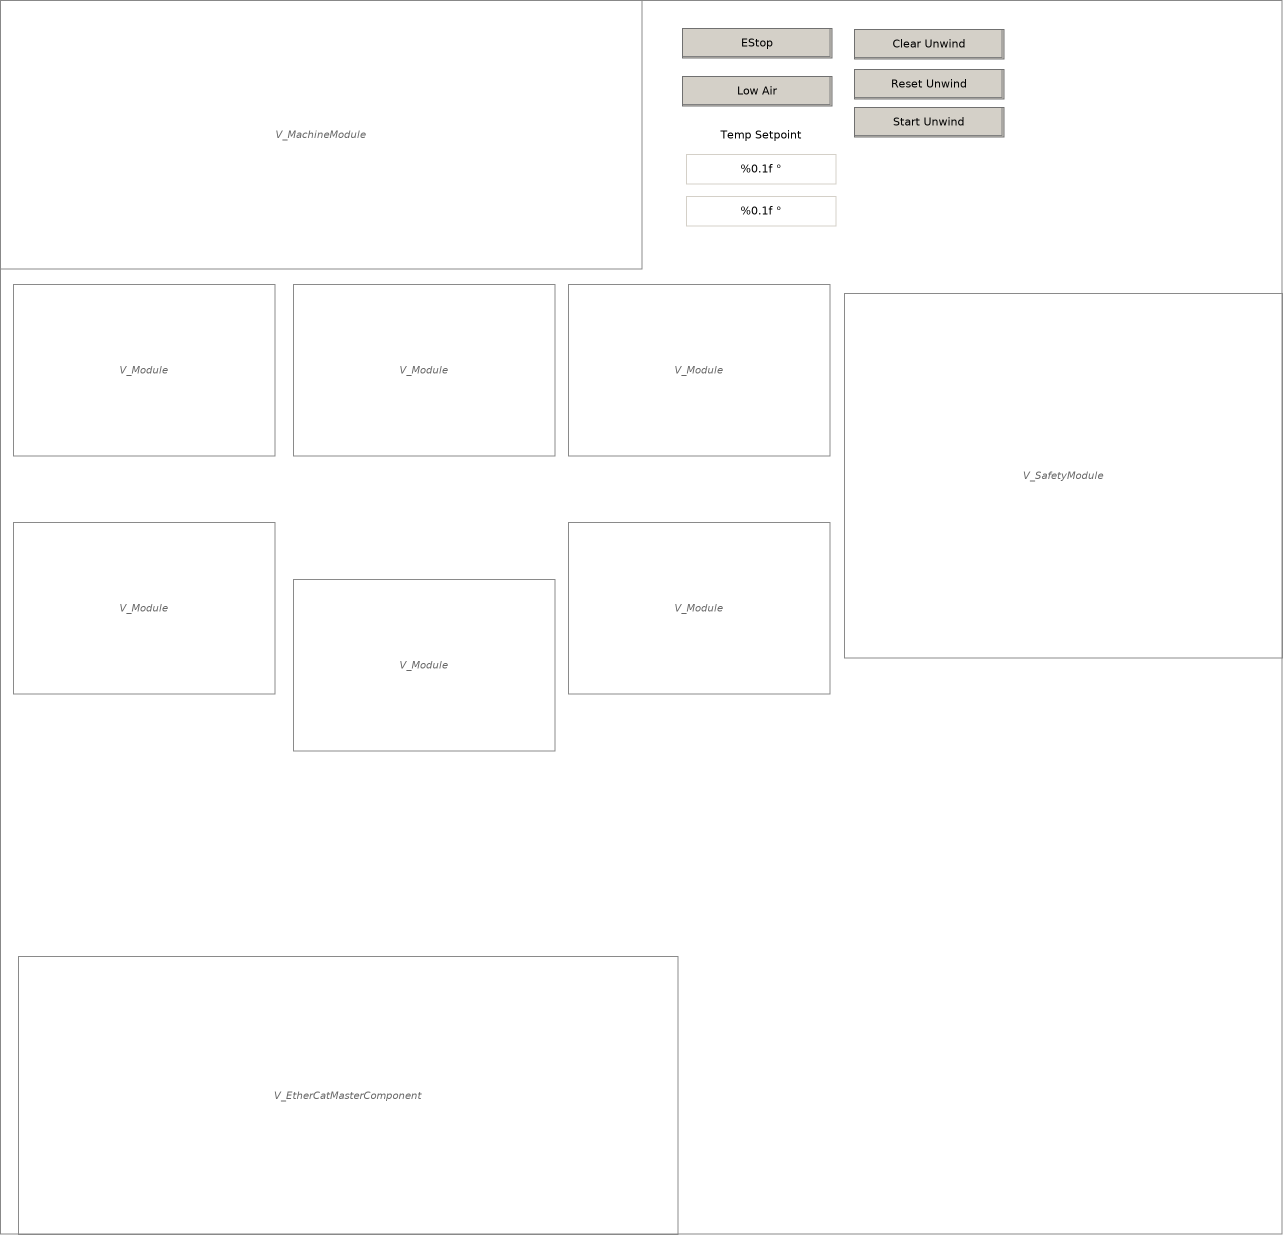
VISUALIZATION V_Main  // 1283x1235
    Frame (0,0 642x269)
        shows V_MachineModule(HMI := MAIN.Machine.PackMLBaseModule_HMI)
    Frame (568,284 262x172)
        shows V_Module(HMI := MAIN.Machine.Station_4.PackMLBaseModule_HMI)
    Frame (568,522 262x172)
        shows V_Module(HMI := MAIN.Machine.Station_5.PackMLBaseModule_HMI)
    Button (682,28 150x30), "EStop"
        toggle MAIN.Machine.EstopInput
    Button (682,76 150x30), "Low Air"
        toggle MAIN.Machine.LowAirInput
    Textfield (686,154 150x30), "%0.1f °", text variable: MAIN.Machine.Sealer.SealBar._SetTemperature
        OnMouseDown: write the text variable via VisuDialogs.Numpad, min 20, max 400, title 'Sealer Bar Temp Setpoint', format %0.1f
    Label (686,120 150x30), "Temp Setpoint"
    Textfield (686,196 150x30), "%0.1f °", text variable: MAIN.Machine.Sealer.SealBar._ActualTemperature
    Button (854,29 150x30), "Clear Unwind"
        OnMouseClick: execute { MAIN.Machine.unwind.PackMLBaseModule_HMI.Command.State := E_PMLCommand.ePMLCommand_Clear; }
    Button (854,69 150x30), "Reset Unwind"
        OnMouseClick: execute { MAIN.Machine.unwind.PackMLBaseModule_HMI.Command.State := E_PMLCommand.ePMLCommand_Reset; }
    Button (854,107 150x30), "Start Unwind"
        OnMouseClick: execute { MAIN.Machine.unwind.PackMLBaseModule_HMI.Command.State := E_PMLCommand.ePMLCommand_Start; }
    Frame (844,293 439x365)
        shows V_SafetyModule(HMI := MAIN.Machine.Safety_SubModule.PackMLBaseModule_HMI)
    Frame (18,956 660x279)
        shows V_EtherCatMasterComponent(EtherCatMaster_HMI := MAIN.Machine.Systems_SubModule.Diagnostics.EtherCatMasterX001.EtherCatMaster_HMI)
    Frame (13,284 262x172)
        shows V_Module(HMI := MAIN.Machine.Station_2.PackMLBaseModule_HMI)
    Frame (293,284 262x172)
        shows V_Module(HMI := MAIN.Machine.Station_3.PackMLBaseModule_HMI)
    Frame (13,522 262x172)
        shows V_Module(HMI := MAIN.Machine.Station_1.PackMLBaseModule_HMI)
    Frame (293,579 262x172)
        shows V_Module(HMI := MAIN.MachineStation_6.PackMLBaseModule_HMI)
END_VISUALIZATION

(* stored: Version 1.1.0.1, ProductVersion 3.1.4024.16
   Visu V_Main: Id {a820fc1e-d71f-479f-a200-f2cc0d18dc0b} *)
